PROGRAM MAIN
VAR CONSTANT
	INSTANCE_NAME: STRING := 'MAIN Program';
	IGNORE_DEFINITION: BOOL := TRUE;
	IGNORE_STOP: BOOL := TRUE;
END_VAR
VAR
	// define services
	m_buttonManager: ButtonManager;
	m_errorManager: ErrorManager;
	m_services: ServiceContainer(ADR(m_errorManager));
	
	// instantiate machine behavior model
	m_container: xPPU_Container(
		m_services.PtrStateTracker, 
		m_services.PtrProcessManager, 
		ADR(m_errorManager));
	
	// INTERLOCKS - must always be False
	// (EProcessVariables.LSC_RampEndWPCount >= 3) AND ((EProcessVariables.LSC_RampStartWPCount >= 3) OR ((EProcessVariables.LSC_RampMiddleWPCount >= 3) OR (EProcessVariables.SSC_RampWPCount >= 3)))
	m_compExpr1: ComparisonExpression(EProcessVariables.LSC_RampEndWPCount, EComparisonType.greater_eq, EDataType.numeric, FALSE, 3, '', TRUE);
	m_compExpr3: ComparisonExpression(EProcessVariables.LSC_RampStartWPCount, EComparisonType.greater_eq, EDataType.numeric, FALSE, 3, '', TRUE);
	m_compExpr5: ComparisonExpression(EProcessVariables.LSC_RampMiddleWPCount, EComparisonType.greater_eq, EDataType.numeric, FALSE, 3, '', TRUE);
	m_compExpr7: ComparisonExpression(EProcessVariables.SSC_RampWPCount, EComparisonType.greater_eq, EDataType.numeric, FALSE, 3, '', TRUE);
	m_boolExpr8: BoolExpression(m_compExpr5, EBoolOperation.or_op, m_compExpr7);
	m_boolExpr9: BoolExpression(m_compExpr3, EBoolOperation.or_op, m_boolExpr8);
	m_allRampsFull: BoolExpression(m_compExpr1, EBoolOperation.and_op, m_boolExpr9);
	
	// INTERLOCKS - must always be True
	// ...
	
	// MANUAL STRATEGY
	m_startAuto: BOOL;
	m_startManual: BOOL;
	m_stopManual: BOOL;
	m_strategyState: EOperationResult;
	
	// other
	i: UINT;
	m_statesEnum: EProcessVariables;
	m_emptyParams: ParameterSet;
	m_didFinishPrimitives: BOOL;
	m_appInitialized: BOOL;
	m_xPPU: xPPU_Automatic;
	m_customSeqStatus: EOperationResult;
	m_steps: ARRAY [0..2] OF STRING;
	m_appObservation: ARRAY[EProcessVariables.operating_mode..EProcessVariables.operating_mode] OF SValue;
	
	// global alarm flags
	m_alarm_flags: ARRAY [1..21] OF BOOL := [FALSE, FALSE, FALSE, FALSE, FALSE, FALSE, FALSE, FALSE, FALSE, FALSE, FALSE, FALSE, FALSE, FALSE, FALSE, FALSE, FALSE, FALSE,FALSE, FALSE]; 
	// global alarm timer
	m_timer_RampStart: TON;
	m_timer_RampMiddle: TON;
	m_timer_PresenceSensor: TON;
	
	m_timer_OpticalSensorStart:TON;
	m_timer_OpticalSensorMid:TON;
	m_timer_OpticalSensorEnd:TON;
	m_timer_InductiveSensorMid:TON;
	m_timer_InductiveSensorStart:TON;
	m_timer_CylinderRampStartExtended :TON;
	m_timer_CylinderRampStartAbnormal :TON;
	m_timer_CylinderRampMidExtended :TON;
	m_timer_CylinderRampMidAbnormal :TON;
	m_timer_PAC_WPAtEnd:TON;
	m_timer_CylinderExtended: TOF;
	m_timer_StackCylinderStuck : TON;
	m_timer_StampSlidingCylinderStuck : TON;
	m_timer_SSC_WPAtEnd : TON;
	m_timer_SSC_WPAtEntry : TON;
	m_timer_RFC_WPAtEntry : TON;
	fb_RFC_SwitchFalling : F_TRIG;   // detect falling edge of RFC switch
   	fb_RFC_WPAtEndFalling    : F_TRIG;   // detect falling edge of RFC_WPAtEnd
  	fb_RFC_WPAtEndRising     : R_TRIG;   // detect rising edge of RFC_WPAtEnd
	
	PreConditon : BOOL;
END_VAR

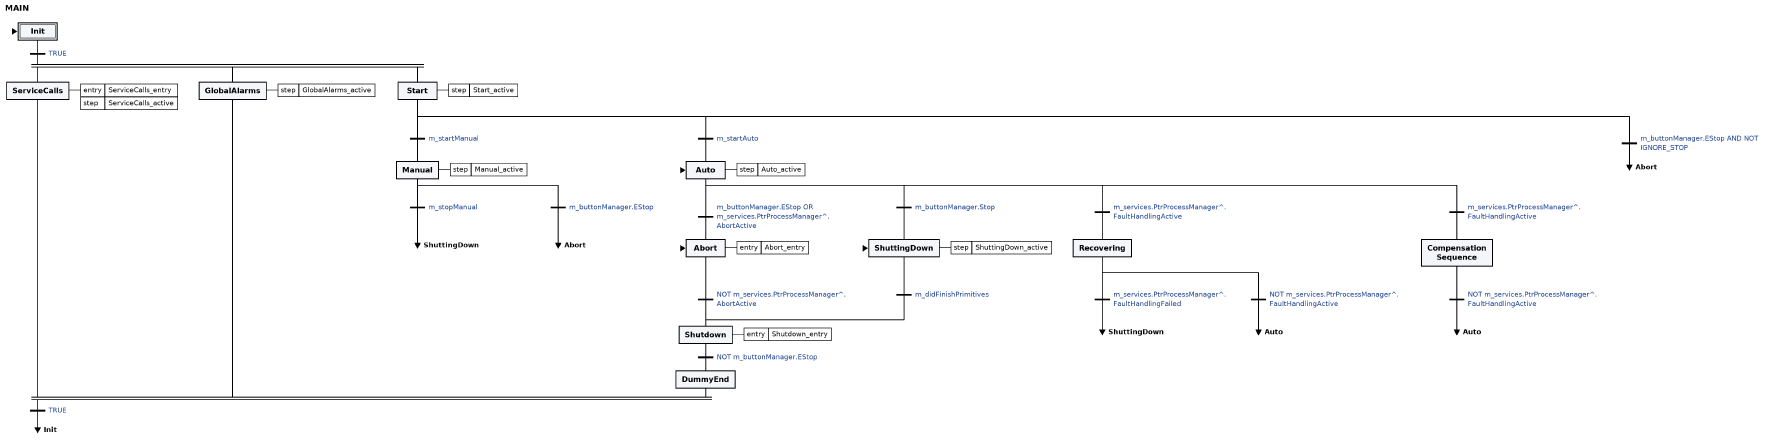
INITIAL_STEP Init:
END_STEP
TRANSITION FROM Init TO (ServiceCalls, GlobalAlarms, Start)
    := TRUE;
END_TRANSITION
STEP ServiceCalls:
    ServiceCalls_entry(P1);  // entry action
    ServiceCalls_active(N);  // step action
END_STEP
STEP GlobalAlarms:
    GlobalAlarms_active(N);  // step action
END_STEP
STEP Start:
    Start_active(N);  // step action
END_STEP
TRANSITION FROM Start TO Manual
    := m_startManual;
END_TRANSITION
STEP Manual:
    Manual_active(N);  // step action
END_STEP
TRANSITION FROM Manual TO ShuttingDown
    := m_stopManual;
END_TRANSITION
TRANSITION FROM Manual TO Abort
    := m_buttonManager.EStop;
END_TRANSITION
TRANSITION FROM Start TO Auto
    := m_startAuto;
END_TRANSITION
STEP Auto:
    Auto_active(N);  // step action
END_STEP
TRANSITION FROM Auto TO Abort
    := m_buttonManager.EStop OR m_services.PtrProcessManager^.AbortActive;
END_TRANSITION
STEP Abort:
    Abort_entry(P1);  // entry action
END_STEP
TRANSITION FROM Abort TO Shutdown
    := NOT m_services.PtrProcessManager^.AbortActive;
END_TRANSITION
TRANSITION FROM Auto TO ShuttingDown
    := m_buttonManager.Stop;
END_TRANSITION
STEP ShuttingDown:
    ShuttingDown_active(N);  // step action
END_STEP
TRANSITION FROM ShuttingDown TO Shutdown
    := m_didFinishPrimitives;
END_TRANSITION
TRANSITION FROM Auto TO Recovering
    := m_services.PtrProcessManager^.FaultHandlingActive;
END_TRANSITION
STEP Recovering:
END_STEP
TRANSITION FROM Recovering TO ShuttingDown
    := m_services.PtrProcessManager^.FaultHandlingFailed;
END_TRANSITION
TRANSITION FROM Recovering TO Auto
    := NOT m_services.PtrProcessManager^.FaultHandlingActive;
END_TRANSITION
TRANSITION FROM Auto TO CompensationSequence
    := m_services.PtrProcessManager^.FaultHandlingActive;
END_TRANSITION
STEP CompensationSequence:
END_STEP
TRANSITION FROM CompensationSequence TO Auto
    := NOT m_services.PtrProcessManager^.FaultHandlingActive;
END_TRANSITION
STEP Shutdown:
    Shutdown_entry(P1);  // entry action
END_STEP
TRANSITION FROM Shutdown TO DummyEnd
    := NOT m_buttonManager.EStop;
END_TRANSITION
TRANSITION FROM Start TO Abort
    := m_buttonManager.EStop AND NOT IGNORE_STOP;
END_TRANSITION
STEP DummyEnd:
END_STEP
TRANSITION FROM (ServiceCalls, GlobalAlarms, DummyEnd) TO Init
    := TRUE;
END_TRANSITION

ACTION Abort_entry:
m_services.PtrProcessManager^.RequestAbort();
END_ACTION

ACTION Auto_active:
m_xPPU(
	i_ptrErrorManager := m_services.PtrErrorManager,
	i_ptrProcessManager := m_services.PtrProcessManager,
	i_ptrStateTracker := m_services.PtrStateTracker);
END_ACTION

ACTION GlobalAlarms_active:
IF m_alarm_flags[1] = FALSE AND m_services.PtrStateTracker^.GetNumeric(EProcessVariables.LSC_RampStartWPCount) = 3 THEN
	m_errorManager.AddMessage(EAlarms.LSC_RampStart_almost_full, TRUE, ESeverity.warning, '3 White WP at Ramp already');
	m_alarm_flags[1] := TRUE;
END_IF

IF m_alarm_flags[2] = FALSE AND m_services.PtrStateTracker^.GetNumeric(EProcessVariables.LSC_RampMiddleWPCount) = 3 THEN
	m_errorManager.AddMessage(EAlarms.LSC_RampMid_almost_full, TRUE, ESeverity.warning, '3 Black WP at Ramp already');
	m_alarm_flags[2] := TRUE;
END_IF

IF m_alarm_flags[3] = FALSE AND m_services.PtrStateTracker^.GetNumeric(EProcessVariables.LSC_RampEndWPCount) = 3 THEN
	m_errorManager.AddMessage(EAlarms.LSC_RampEnd_almost_full, TRUE, ESeverity.warning, '3 Unknown WP at Ramp already');
	m_alarm_flags[3] := TRUE;
END_IF

IF m_alarm_flags[1] = FALSE AND m_services.PtrStateTracker^.GetNumeric(EProcessVariables.LSC_RampStartWPCount) > 3 THEN
	m_errorManager.AddMessage(EAlarms.LSC_RampStart_full, TRUE, ESeverity.error, 'More than 3 White WP at Ramp');
	m_alarm_flags[1] := TRUE;
END_IF

IF m_alarm_flags[2] = FALSE AND m_services.PtrStateTracker^.GetNumeric(EProcessVariables.LSC_RampMiddleWPCount) > 3 THEN
	m_errorManager.AddMessage(EAlarms.LSC_RampMid_full, TRUE, ESeverity.error, 'More than 3 Black WP at Ramp');
	m_alarm_flags[2] := TRUE;
END_IF

IF m_alarm_flags[3] = FALSE AND m_services.PtrStateTracker^.GetNumeric(EProcessVariables.LSC_RampEndWPCount) > 3 THEN
	m_errorManager.AddMessage(EAlarms.LSC_RampEnd_full, TRUE, ESeverity.error, 'More than 3 Unknown WP at Ramp');
	m_alarm_flags[3] := TRUE;
END_IF
// new alarm
m_timer_PresenceSensor(IN := m_services.PtrStateTracker^.GetBinary(EProcessVariables.LSC_WorkpieceAtEntry), PT := T#3000MS);
IF m_alarm_flags[4] = FALSE AND m_timer_PresenceSensor.Q  
	THEN
	m_errorManager.AddMessage(EAlarms.LSC_Entry_accumulated, TRUE, ESeverity.error, 'WP accumulated at Entry on LSC');
	m_timer_PresenceSensor(IN := FALSE);
	m_alarm_flags[4] := TRUE;
END_IF

m_timer_OpticalSensorStart(IN := m_services.PtrStateTracker^.GetBinary(EProcessVariables.LSC_LightWPAtStart), PT := T#3000MS);
m_timer_InductiveSensorStart(IN := m_services.PtrStateTracker^.GetBinary(EProcessVariables.LSC_MetalWPAtStart), PT := T#3000MS);
IF m_alarm_flags[5] = FALSE AND (m_timer_OpticalSensorStart.Q OR m_timer_InductiveSensorStart.Q)
    THEN
	m_errorManager.AddMessage(EAlarms.LSC_FirstPairOfSensors_accumulated, TRUE, ESeverity.error, 'WP accmulated at the first pair of sensors on LSC');
	m_timer_OpticalSensorStart(IN := FALSE);
	m_alarm_flags[5] := TRUE;
END_IF

m_timer_OpticalSensorMid(IN := m_services.PtrStateTracker^.GetBinary(EProcessVariables.LSC_MetalWPAtMid), PT := T#3000MS);
m_timer_InductiveSensorMid(IN := m_services.PtrStateTracker^.GetBinary(EProcessVariables.LSC_LightWPAtMid), PT := T#3000MS);
IF m_alarm_flags[6] = FALSE AND (m_timer_OpticalSensorMid.Q OR m_timer_InductiveSensorMid.Q) 
   THEN
	m_errorManager.AddMessage(EAlarms.LSC_SecondPairOfSensors_accumulated, TRUE, ESeverity.error, 'WP accmulated at Middle on LSC');
	m_timer_OpticalSensorMid(IN := FALSE);
	m_alarm_flags[6] := TRUE;
END_IF


m_timer_OpticalSensorEnd(IN := m_services.PtrStateTracker^.GetBinary(EProcessVariables.LSC_LightWPAtEnd), PT := T#3000MS);
IF m_alarm_flags[7] = FALSE AND m_timer_OpticalSensorEnd.Q 
   THEN
	m_errorManager.AddMessage(EAlarms.LSC_End_accumulated, TRUE, ESeverity.error, 'WP accmulated at End on LSC');
	m_timer_OpticalSensorEnd(IN := FALSE);
	m_alarm_flags[7] := TRUE;
END_IF

IF m_alarm_flags[8] = FALSE 
	AND m_services.PtrStateTracker^.GetBinary(EProcessVariables.Stack_CylinderExtended)
	AND m_services.PtrStateTracker^.GetNumeric(EProcessVariables.Stack_WPWeight) < 1500
THEN
	m_errorManager.AddMessage(EAlarms.stack_no_WP, TRUE, ESeverity.warning, 'No WP in Magazine');
	m_alarm_flags[8] := TRUE; 
END_IF

m_timer_CylinderRampStartExtended(IN := m_services.PtrStateTracker^.GetBinary(EProcessVariables.LSC_CylinderRampStartExtended), PT := T#3000MS);
IF m_alarm_flags[9] = FALSE
	AND m_timer_CylinderRampStartExtended.Q
THEN
	m_errorManager.AddMessage(EAlarms.LSC_RampStart_wrong_eject, TRUE, ESeverity.error, 'WP was not corretly pushed into RampStart');
	m_alarm_flags[9] := TRUE;
END_IF

m_timer_CylinderRampMidExtended(IN := m_services.PtrStateTracker^.GetBinary(EProcessVariables.LSC_CylinderRampMidExtended), PT := T#3000MS);
IF m_alarm_flags[10] = FALSE
	AND m_timer_CylinderRampMidExtended.Q
THEN
	m_errorManager.AddMessage(EAlarms.LSC_RampMid_wrong_eject, TRUE, ESeverity.error, 'WP was not corretly pushed into RampMid');
	m_alarm_flags[10] := TRUE;
END_IF

//New alarm
PreConditon:= m_services.PtrStateTracker^.GetBinary(EProcessVariables.PAC_WPAtEnd) AND NOT m_services.PtrStateTracker^.GetBinary(EProcessVariables.SSC_WPAtStart);
m_timer_PAC_WPAtEnd(IN := PreConditon, PT := T#6000MS);
IF m_alarm_flags[11] = FALSE AND m_timer_PAC_WPAtEnd.Q 
   THEN
	m_errorManager.AddMessage(EAlarms.LSC_End_accumulated, TRUE, ESeverity.error, 'WP accmulated at End on PAC');
	m_timer_OpticalSensorEnd(IN := FALSE);
	m_alarm_flags[11] := TRUE;
END_IF

m_timer_CylinderRampStartAbnormal(IN := (NOT m_services.PtrStateTracker^.GetBinary(EProcessVariables.LSC_CylinderRampStartExtended))
									AND (NOT m_services.PtrStateTracker^.GetBinary(EProcessVariables.LSC_CylinderRampStartRetracted)), PT := T#3000MS);
IF m_alarm_flags[12] = FALSE AND m_timer_CylinderRampStartAbnormal.Q
   THEN
	m_errorManager.AddMessage(EAlarms.LSC_Cylinder1_abnormal, TRUE, ESeverity.error, 'The pushing cylinder at the entry is abnormal');
	m_timer_OpticalSensorEnd(IN := FALSE);
	m_alarm_flags[12] := TRUE;
END_IF

m_timer_CylinderRampMidAbnormal(IN := (NOT m_services.PtrStateTracker^.GetBinary(EProcessVariables.LSC_CylinderRampMidExtended))
									AND (NOT m_services.PtrStateTracker^.GetBinary(EProcessVariables.LSC_CylinderRampMidRetracted)), PT := T#3000MS);
IF m_alarm_flags[13] = FALSE AND m_timer_CylinderRampMidAbnormal.Q
   THEN
	m_errorManager.AddMessage(EAlarms.LSC_Cylinder2_abnormal, TRUE, ESeverity.error, 'The pushing cylinder in the middle is abnormal');
	m_timer_OpticalSensorEnd(IN := FALSE);
	m_alarm_flags[13] := TRUE;
END_IF

m_timer_StackCylinderStuck(IN := (NOT m_services.PtrStateTracker^.GetBinary(EProcessVariables.Stack_CylinderExtended)) 
                          AND (NOT m_services.PtrStateTracker^.GetBinary(EProcessVariables.Stack_CylinderRetracted)), PT := T#3000MS);
IF m_alarm_flags[14] = FALSE
	AND m_services.PtrStateTracker^.GetBinary(EProcessVariables.Stack_WorkpieceAvailable)
	AND m_timer_StackCylinderStuck.Q
THEN
	m_errorManager.AddMessage(EAlarms.stack_WP_stuck,TRUE, ESeverity.error, 'WP stuck at pick up station');
	m_alarm_flags[14] := TRUE;
END_IF

m_timer_StampSlidingCylinderStuck(IN := (NOT m_services.PtrStateTracker^.GetBinary(EProcessVariables.Stamp_SlidingCylinderExtended)) 
                          AND (NOT m_services.PtrStateTracker^.GetBinary(EProcessVariables.Stamp_SlidingCylinderRetracted)), PT := T#3000MS);
IF m_alarm_flags[15] = FALSE
	AND m_timer_StampSlidingCylinderStuck.Q
THEN
	m_errorManager.AddMessage(EAlarms.stamp_SlidingCylinder_stuck,TRUE, ESeverity.error, 'Stamp SlidingCylinder is stuck');
	m_alarm_flags[15] := TRUE;
END_IF

m_timer_SSC_WPAtEnd(IN := m_services.PtrStateTracker^.GetBinary(EProcessVariables.SSC_WPAtEnd), PT := T#3000MS);
IF m_alarm_flags[16] = FALSE AND m_timer_SSC_WPAtEnd.Q 
   THEN
	m_errorManager.AddMessage(EAlarms.SSC_End_accumulated, TRUE, ESeverity.error, 'WP accmulated at End on SSC');
	m_timer_OpticalSensorEnd(IN := FALSE);
	m_alarm_flags[16] := TRUE;
END_IF

m_timer_SSC_WPAtEntry(IN := m_services.PtrStateTracker^.GetBinary(EProcessVariables.SSC_WPAtStart), PT := T#3000MS);
IF m_alarm_flags[17] = FALSE AND m_timer_SSC_WPAtEntry.Q  
	THEN
	m_errorManager.AddMessage(EAlarms.SSC_Entry_accumulated, TRUE, ESeverity.error, 'WP accumulated at Entry on SSC');
	m_timer_SSC_WPAtEntry(IN := FALSE);
	m_alarm_flags[17] := TRUE;
END_IF

m_timer_RFC_WPAtEntry(IN := m_services.PtrStateTracker^.GetBinary(EProcessVariables.RFC_WPAtStart), PT := T#3000MS);
IF m_alarm_flags[18] = FALSE AND m_timer_RFC_WPAtEntry.Q  
	THEN
	m_errorManager.AddMessage(EAlarms.RFC_Entry_accumulated, TRUE, ESeverity.error, 'WP accumulated at Entry on RFC');
	m_timer_RFC_WPAtEntry(IN := FALSE);
	m_alarm_flags[18] := TRUE;
END_IF

//new alarm
fb_RFC_SwitchFalling(CLK := m_services.PtrStateTracker^.GetBinary(EProcessVariables.RFC_SwitchExtended));
fb_RFC_WPAtEndFalling(CLK := m_services.PtrStateTracker^.GetBinary(EProcessVariables.RFC_WPAtEnd));
fb_RFC_WPAtEndRising(CLK := m_services.PtrStateTracker^.GetBinary(EProcessVariables.RFC_WPAtEnd));
// If switch falls and RFC_WPAtEnd remains true with no change, set alarm
IF m_alarm_flags[19] = FALSE AND fb_RFC_SwitchFalling.Q 
   AND (m_services.PtrStateTracker^.GetBinary(EProcessVariables.RFC_WPAtEnd))  // RFC_WPAtEnd is still true
   AND NOT fb_RFC_WPAtEndFalling.Q  // no falling edge on RFC_WPAtEnd
   AND NOT fb_RFC_WPAtEndRising.Q   // no rising edge on RFC_WPAtEnd
THEN
	m_errorManager.AddMessage(EAlarms.RFC_End_accumulated, TRUE, ESeverity.error, 'WP accumulated at End on RFC');
   	m_alarm_flags[19] := TRUE;
END_IF

IF m_alarm_flags[20] = FALSE AND m_services.PtrStateTracker^.GetNumeric(EProcessVariables.SSC_RampWPCount) = 3 THEN
	m_errorManager.AddMessage(EAlarms.SSC_RampEnd_almost_full, TRUE, ESeverity.warning, '3 WP at Ramp of SSC already');
	m_alarm_flags[20] := TRUE;
END_IF

IF m_alarm_flags[21] = FALSE AND m_services.PtrStateTracker^.GetNumeric(EProcessVariables.SSC_RampWPCount) > 3 THEN
	m_errorManager.AddMessage(EAlarms.SSC_Ramp_full, TRUE, ESeverity.error, 'More than 3 WP at Ramp of SSC');
	m_alarm_flags[21] := TRUE;
END_IF


//m_timer_CylinderExtended(IN := (m_services.PtrStateTracker^.GetBinary(EProcessVariables.Crane_AtStack) AND m_services.PtrStateTracker^.GetBinary(EProcessVariables.Crane_CylinderExtended)), PT:=T#500MS);
//IF m_alarm_flags[7] = FALSE AND m_timer_CylinderExtended.Q = TRUE AND m_services.PtrStateTracker^.GetBinary(EProcessVariables.Crane_HoldingWorkpiece) = FALSE AND m_services.PtrStateTracker^.GetBinary(EProcessVariables.Crane_CylinderRetracted) AND m_services.PtrStateTracker^.GetBinary(EProcessVariables.Stack_WorkpieceAvailable) THEN
	//m_errorManager.AddMessage(EAlarms.crane_gripper_failed, TRUE, ESeverity.error, 'crane failed to pick up WP at Stack');
 	//m_alarm_flags[7] := TRUE;
//END_IF


//IF m_services.PtrStateTracker^.GetBinary(EProcessVariables.Crane_AtStack) 
//	AND m_services.PtrStateTracker^.GetNumeric(EProcessVariables.LSC_ProductType) = 1 THEN
//	m_errorManager.AddMessage(EAlarms.changs_alarm, TRUE, ESeverity.error, 'GlobalAlarms');
//END_IF

//Stack #1
//IF m_services.PtrStateTracker^.GetNumeric(EProcessVariables.Stack_ProductType) = EProductTypes.none
	//AND m_services.PtrStateTracker^.GetBinary(EProcessVariables.Stack_WorkpieceAvailable) THEN
	//m_errorManager.AddMessage(EAlarms.WPupdate_wrong, TRUE, ESeverity.error, 'Stack_GlobalAlarms');
//END_IF

//Stack - Crane #1
//IF m_services.PtrStateTracker^.GetBinary(EProcessVariables.Crane_AtStack) 
//	AND m_services.PtrStateTracker^.GetBinary(EProcessVariables.Crane_HoldingWorkpiece) 
  //  AND m_services.PtrStateTracker^.GetBinary(EProcessVariables.Crane_CylinderRetracted) 
  //  AND m_services.PtrStateTracker^.GetBinary(EProcessVariables.Stack_WorkpieceAvailable) THEN
	//m_errorManager.AddMessage(EAlarms.stack_occupied, TRUE, ESeverity.warning, 'stack_GlobalAlarms');
//END_IF

//Crane #1  
//IF m_services.PtrStateTracker^.GetBinary(EProcessVariables.Crane_CylinderExtended) 
	//AND m_services.PtrStateTracker^.GetBinary(EProcessVariables.Crane_CylinderRetracted) THEN
	//m_errorManager.AddMessage(EAlarms.changs_alarm, TRUE, ESeverity.error, 'GlobalAlarms');
//END_IF

//Crane - Stamp #1
//IF m_services.PtrStateTracker^.GetBinary(EProcessVariables.Crane_AtStamp) 
//	AND m_services.PtrStateTracker^.GetBinary(EProcessVariables.Crane_HoldingWorkpiece) 
//	AND m_services.PtrStateTracker^.GetBinary(EProcessVariables.Crane_CylinderRetracted) 
//	AND m_services.PtrStateTracker^.GetBinary(EProcessVariables.Stamp_WPAtStamp) THEN
//	m_errorManager.AddMessage(EAlarms.changs_alarm, TRUE, ESeverity.error, 'GlobalAlarms');
//END_IF

// Stamp #1
//IF   m_services.PtrStateTracker^.GetBinary(EProcessVariables.Stamp_WPAtStamp)
//AND (m_services.PtrStateTracker^.GetNumeric(EProcessVariables.Stamp_WorkpieceState) = EStampStates.none
//OR  m_services.PtrStateTracker^.GetNumeric(EProcessVariables.Stamp_ProductType) = EProductTypes.none) THEN
	//m_errorManager.AddMessage(EAlarms.WPupdate_wrong, TRUE, ESeverity.error, 'Stamp_GlobalAlarms');
//END_IF

// Stamp #1
//IF m_services.PtrStateTracker^.GetNumeric(EProcessVariables.Stamp_WorkpieceState) = EStampStates.pressed
//	AND  m_services.PtrStateTracker^.GetBinary(EProcessVariables.Stamp_WPAtStamp) THEN
//	m_errorManager.AddMessage(EAlarms.changs_alarm, TRUE, ESeverity.error, 'GlobalAlarms');
//END_IF

// Crane - LSC #1
//IF m_services.PtrStateTracker^.GetBinary(EProcessVariables.LSC_WorkpieceAtEntry) 
//	AND m_services.PtrStateTracker^.GetBinary(EProcessVariables.Crane_HoldingWorkpiece) 
	//AND m_services.PtrStateTracker^.GetBinary(EProcessVariables.Crane_CylinderRetracted) 
//	AND m_services.PtrStateTracker^.GetBinary(EProcessVariables.LSC_WorkpieceAtEntry) THEN
	//m_errorManager.AddMessage(EAlarms.changs_alarm, TRUE, ESeverity.error, 'GlobalAlarms');
//END_IF

// LSC #1
//IF m_services.PtrStateTracker^.GetBinary(EProcessVariables.LSC_WorkpieceAtEntry) 
	//AND ((m_services.PtrStateTracker^.GetNumeric(EProcessVariables.LSC_ProductType) = 1)
	//OR (m_services.PtrStateTracker^.GetNumeric(EProcessVariables.LSC_ProductType) = 2)
//(m_services.PtrStateTracker^.GetNumeric(EProcessVariables.LSC_ProductType) = 3)
 // OR (m_services.PtrStateTracker^.GetNumeric(EProcessVariables.LSC_ProductType) = 4)) THEN
	//m_errorManager.AddMessage(EAlarms.changs_alarm, TRUE, ESeverity.error, 'GlobalAlarms');
//END_IF
END_ACTION

ACTION Manual_active:


m_strategyState := m_services.PtrProcessManager^.ExecuteCustomStrategy();
m_stopManual := m_buttonManager.Stop 
	OR NOT m_services.PtrProcessManager^.CustomStrategyReady 
	OR m_strategyState = EOperationResult.success;
END_ACTION

ACTION ServiceCalls_active:
// process state observation
m_appObservation[EProcessVariables.operating_mode].DataType := EDataType.string_t;
m_appObservation[EProcessVariables.operating_mode].Value.String_t := SFCCurrentStep;

// cylic service updates
IF m_services.PtrStateTracker <>0 THEN
m_services.PtrStateTracker^.CyclicUpdateStatus(IGNORE_DEFINITION,m_appObservation);
m_services.PtrProcessManager^.CyclicManageBehavior();
END_IF
END_ACTION

ACTION ServiceCalls_dummy:
IF m_alarm_flags[1] = FALSE AND m_services.PtrStateTracker^.GetNumeric(EProcessVariables.LSC_RampStartWPCount) = 3 THEN
	m_errorManager.AddMessage(EAlarms.LSC_RampStart_almost_full, TRUE, ESeverity.warning, '3 White WP at Ramp already');
	m_alarm_flags[1] := TRUE;
END_IF

IF m_alarm_flags[2] = FALSE AND m_services.PtrStateTracker^.GetNumeric(EProcessVariables.LSC_RampMiddleWPCount) = 3 THEN
	m_errorManager.AddMessage(EAlarms.LSC_RampMid_almost_full, TRUE, ESeverity.warning, '3 Black WP at Ramp already');
	m_alarm_flags[2] := TRUE;
END_IF

IF m_alarm_flags[3] = FALSE AND m_services.PtrStateTracker^.GetNumeric(EProcessVariables.LSC_RampEndWPCount) = 3 THEN
	m_errorManager.AddMessage(EAlarms.LSC_RampEnd_almost_full, TRUE, ESeverity.warning, '3 Unknown WP at Ramp already');
	m_alarm_flags[3] := TRUE;
END_IF

IF m_alarm_flags[1] = TRUE AND m_services.PtrStateTracker^.GetNumeric(EProcessVariables.LSC_RampStartWPCount) > 3 THEN
	m_errorManager.AddMessage(EAlarms.LSC_RampStart_full, TRUE, ESeverity.error, 'More than 3 White WP at Ramp');
	m_alarm_flags[1] := FALSE;
END_IF

IF m_alarm_flags[2] = TRUE AND m_services.PtrStateTracker^.GetNumeric(EProcessVariables.LSC_RampMiddleWPCount) > 3 THEN
	m_errorManager.AddMessage(EAlarms.LSC_RampStart_full, TRUE, ESeverity.error, 'More than 3 Black WP at Ramp');
	m_alarm_flags[2] := FALSE;
END_IF

IF m_alarm_flags[3] = TRUE AND m_services.PtrStateTracker^.GetNumeric(EProcessVariables.LSC_RampEndWPCount) > 3 THEN
	m_errorManager.AddMessage(EAlarms.LSC_RampStart_full, TRUE, ESeverity.error, 'More than 3 Unknown WP at Ramp');
	m_alarm_flags[3] := FALSE;
END_IF

m_timer_PresenceSensor(IN := m_services.PtrStateTracker^.GetBinary(EProcessVariables.LSC_WorkpieceAtEntry), PT := T#3000MS);
IF m_alarm_flags[4] = FALSE AND m_timer_PresenceSensor.Q  
	THEN
	m_errorManager.AddMessage(EAlarms.LSC_Entry_accumulated, TRUE, ESeverity.error, 'WP accmulated at Entry on LSC');
	m_timer_PresenceSensor(IN := FALSE);
	m_alarm_flags[4] := TRUE;
END_IF

m_timer_OpticalSensorStart(IN := m_services.PtrStateTracker^.GetBinary(EProcessVariables.LSC_WPAtRampStart), PT := T#3000MS);
IF m_alarm_flags[5] = FALSE AND m_timer_RampStart.Q
    THEN
	m_errorManager.AddMessage(EAlarms.LSC_FirstPairOfSensors_accumulated, TRUE, ESeverity.error, 'WP accmulated at the first pair of sensors on LSC');
	m_timer_RampStart(IN := FALSE);
	m_alarm_flags[5] := TRUE;
END_IF

m_timer_RampMiddle(IN := m_services.PtrStateTracker^.GetBinary(EProcessVariables.LSC_WPAtRampMiddle), PT := T#3000MS);
IF m_alarm_flags[6] = FALSE AND m_timer_RampMiddle.Q 
   THEN
	m_errorManager.AddMessage(EAlarms.LSC_SecondPairOfSensors_accumulated, TRUE, ESeverity.error, 'WP accmulated at Middle on LSC');
	m_timer_RampMiddle(IN := FALSE);
	m_alarm_flags[6] := TRUE;
END_IF


//IF m_services.PtrStateTracker^.GetBinary(EProcessVariables.Crane_AtStack) 
//	AND m_services.PtrStateTracker^.GetNumeric(EProcessVariables.LSC_ProductType) = 1 THEN
//	m_errorManager.AddMessage(EAlarms.changs_alarm, TRUE, ESeverity.error, 'GlobalAlarms');
//END_IF

//Stack #1
//IF m_services.PtrStateTracker^.GetNumeric(EProcessVariables.Stack_ProductType) = EProductTypes.none
	//AND m_services.PtrStateTracker^.GetBinary(EProcessVariables.Stack_WorkpieceAvailable) THEN
	//m_errorManager.AddMessage(EAlarms.WPupdate_wrong, TRUE, ESeverity.error, 'Stack_GlobalAlarms');
//END_IF

//Stack - Crane #1
//IF m_services.PtrStateTracker^.GetBinary(EProcessVariables.Crane_AtStack) 
//	AND m_services.PtrStateTracker^.GetBinary(EProcessVariables.Crane_HoldingWorkpiece) 
  //  AND m_services.PtrStateTracker^.GetBinary(EProcessVariables.Crane_CylinderRetracted) 
  //  AND m_services.PtrStateTracker^.GetBinary(EProcessVariables.Stack_WorkpieceAvailable) THEN
	//m_errorManager.AddMessage(EAlarms.stack_occupied, TRUE, ESeverity.warning, 'stack_GlobalAlarms');
//END_IF

//Crane #1  
//IF m_services.PtrStateTracker^.GetBinary(EProcessVariables.Crane_CylinderExtended) 
	//AND m_services.PtrStateTracker^.GetBinary(EProcessVariables.Crane_CylinderRetracted) THEN
	//m_errorManager.AddMessage(EAlarms.changs_alarm, TRUE, ESeverity.error, 'GlobalAlarms');
//END_IF

//Crane - Stamp #1
//IF m_services.PtrStateTracker^.GetBinary(EProcessVariables.Crane_AtStamp) 
//	AND m_services.PtrStateTracker^.GetBinary(EProcessVariables.Crane_HoldingWorkpiece) 
//	AND m_services.PtrStateTracker^.GetBinary(EProcessVariables.Crane_CylinderRetracted) 
//	AND m_services.PtrStateTracker^.GetBinary(EProcessVariables.Stamp_WPAtStamp) THEN
//	m_errorManager.AddMessage(EAlarms.changs_alarm, TRUE, ESeverity.error, 'GlobalAlarms');
//END_IF

// Stamp #1
//IF   m_services.PtrStateTracker^.GetBinary(EProcessVariables.Stamp_WPAtStamp)
//AND (m_services.PtrStateTracker^.GetNumeric(EProcessVariables.Stamp_WorkpieceState) = EStampStates.none
//OR  m_services.PtrStateTracker^.GetNumeric(EProcessVariables.Stamp_ProductType) = EProductTypes.none) THEN
	//m_errorManager.AddMessage(EAlarms.WPupdate_wrong, TRUE, ESeverity.error, 'Stamp_GlobalAlarms');
//END_IF

// Stamp #1
//IF m_services.PtrStateTracker^.GetNumeric(EProcessVariables.Stamp_WorkpieceState) = EStampStates.pressed
//	AND  m_services.PtrStateTracker^.GetBinary(EProcessVariables.Stamp_WPAtStamp) THEN
//	m_errorManager.AddMessage(EAlarms.changs_alarm, TRUE, ESeverity.error, 'GlobalAlarms');
//END_IF

// Crane - LSC #1
//IF m_services.PtrStateTracker^.GetBinary(EProcessVariables.LSC_WorkpieceAtEntry) 
//	AND m_services.PtrStateTracker^.GetBinary(EProcessVariables.Crane_HoldingWorkpiece) 
	//AND m_services.PtrStateTracker^.GetBinary(EProcessVariables.Crane_CylinderRetracted) 
//	AND m_services.PtrStateTracker^.GetBinary(EProcessVariables.LSC_WorkpieceAtEntry) THEN
	//m_errorManager.AddMessage(EAlarms.changs_alarm, TRUE, ESeverity.error, 'GlobalAlarms');
//END_IF

// LSC #1
//IF m_services.PtrStateTracker^.GetBinary(EProcessVariables.LSC_WorkpieceAtEntry) 
	//AND ((m_services.PtrStateTracker^.GetNumeric(EProcessVariables.LSC_ProductType) = 1)
	//OR (m_services.PtrStateTracker^.GetNumeric(EProcessVariables.LSC_ProductType) = 2)
//(m_services.PtrStateTracker^.GetNumeric(EProcessVariables.LSC_ProductType) = 3)
 // OR (m_services.PtrStateTracker^.GetNumeric(EProcessVariables.LSC_ProductType) = 4)) THEN
	//m_errorManager.AddMessage(EAlarms.changs_alarm, TRUE, ESeverity.error, 'GlobalAlarms');
//END_IF
END_ACTION

ACTION ServiceCalls_entry:
IF NOT m_appInitialized THEN
	FC_InitAlarmTexts();
	
	// init process variable names
	FOR i := ResiConst.ARR_MIN TO ResiConst.STATE_ARR_MAX DO
		m_statesEnum := i;
		m_services.PtrStateTracker^.SetProcessVariableName(i, TO_STRING(m_statesEnum));
	END_FOR
	
	// add interlocks
	m_services.PtrStateTracker^.AddInterlock(m_allRampsFull, FALSE);
	
	m_appInitialized := TRUE;
	m_errorManager.AddMessage(EAlarms.initialized, TRUE, ESeverity.info, 'MAIN');
END_IF
END_ACTION

ACTION Shutdown_entry:
m_errorManager.AddMessage(
	i_alarmId := EAlarms.stopped,
	i_active := TRUE,
	i_severity := ESeverity.info,
	i_instanceName := INSTANCE_NAME);

m_services.PtrStateTracker^.ResetDefinitions();
END_ACTION

ACTION ShuttingDown_active:
m_didFinishPrimitives := m_services.PtrProcessManager^.FinishPrimitives(i_abortRecoveries := TRUE);
END_ACTION

ACTION Start_active:
m_startManual := m_buttonManager.Mode = EOperatingModes.manual AND m_services.PtrProcessManager^.CustomStrategyReady AND m_buttonManager.Start;
m_startAuto := m_buttonManager.Mode = EOperatingModes.automatic AND m_buttonManager.Start;
END_ACTION

END_PROGRAM

(* stored: Version 1.1.0.1
   POU MAIN: Id {a58bb666-43ab-46d1-86a0-bca8bb16f09d}, SpecialFunc None
   Action Abort_entry: Id {99ab6845-5539-4711-8874-815ac3457b5b}
   Action Auto_active: Id {04ce01cc-9c38-475b-8a5a-1fc20fe7563e}
   Action GlobalAlarms_active: Id {dfa51d6e-f1b0-4c94-9554-ce2b7223f2d9}
   Action Manual_active: Id {2d822a92-05f0-432c-a5a6-99bb4d17c0ba}
   Action ServiceCalls_active: Id {6606d316-b039-41b0-bf6b-5c561aa539c7}
   Action ServiceCalls_dummy: Id {881221eb-adc3-431a-8359-788cd62809a7}
   Action ServiceCalls_entry: Id {24c536b4-2fb2-44ef-8d75-892e48d5ec1d}
   Action Shutdown_entry: Id {056f07e9-48aa-4c4b-bb7b-3ccbd0dcc4b7}
   Action ShuttingDown_active: Id {b1b16c20-54da-4d9f-88a1-e95076766694}
   Action Start_active: Id {edc2770b-bafe-4378-a54c-e488f6b79a86} *)
